INTERFACE I_AdsSymbolProvider EXTENDS __SYSTEM.IQueryInterface

METHOD M_GetAdsSymbolMetadata : BOOL
VAR_OUTPUT
	Address : PVOID;
	Size : UDINT;
END_VAR
END_METHOD

END_INTERFACE

(* stored: Version 1.1.0.1, ProductVersion 3.1.4026.18
   Itf I_AdsSymbolProvider: Id {4cd1d14e-87eb-418a-b098-5ff22d172d55}
   Method M_GetAdsSymbolMetadata: Id {d2bb261d-3ba0-42c1-ac00-7071b4b599f7} *)
